// TIA Portal project "FactoryIO_Template_S7-1500_V15_V16" (V16)

(* hardware
DEVICE "S71500/ET200MP-Station_1"  S7-1500 station
   slot 0: "Profilschiene_0"  6ES7 590-1***0-0AA0
   slot 1: "PLC_1"  CPU 1511-1 PN  6ES7 511-1AK00-0AB0  V1.8
   slot 2: "AI 8xU/I/RTD/TC ST_1"  AI 8xU/I/RTD/TC ST  6ES7 531-7KF00-0AB0  V2.0
   slot 3: "AI 8xU/I/RTD/TC ST_2"  AI 8xU/I/RTD/TC ST  6ES7 531-7KF00-0AB0  V2.0
   slot 4: "AI 8xU/I/RTD/TC ST_3"  AI 8xU/I/RTD/TC ST  6ES7 531-7KF00-0AB0  V2.0
   slot 5: "AI 8xU/I/RTD/TC ST_4"  AI 8xU/I/RTD/TC ST  6ES7 531-7KF00-0AB0  V2.0
   slot 6: "DI 16x24VDC BA_1"  DI 16x24VDC BA  6ES7 521-1BH10-0AA0  V1.0
*)

// ===== PLC "PLC_1"  CPU 1511-1 PN =====

VAR_GLOBAL   // PLC tag table "Standard-Variablentabelle"
   "start" AT %E0.0 : Bool;
   "stop" AT %I0.1 : Bool;
   "vsensör" AT %I0.2 : Bool;
   "konveyor1" AT %Q0.0 : Bool;
   "konveyor2" AT %Q0.1 : Bool;
   "itme" AT %Q0.2 : Bool;
   "yr" AT %M0.0 : Bool;
   "itmebant" AT %Q0.3 : Bool;
   "konveyor3" AT %Q0.4 : Bool;
   "itme2" AT %Q0.5 : Bool;
   "itme2bant" AT %Q0.6 : Bool;
   "vsensör2" AT %I0.3 : Bool;
END_VAR

// folder: System blocks/Program resources

DATA_BLOCK "dzr2"   // DB1
{ S7_Optimized_Access := 'TRUE' }
AUTHOR : Simatic
FAMILY : IEC
NAME : IEC_TMR
VERSION : 1.0
// stored: InstanceOfName IEC_TIMER
"IEC_TIMER"
BEGIN
END_DATA_BLOCK

DATA_BLOCK "dzr3"   // DB2
{ S7_Optimized_Access := 'TRUE' }
AUTHOR : Simatic
FAMILY : IEC
NAME : IEC_TMR
VERSION : 1.0
// stored: InstanceOfName IEC_TIMER
"IEC_TIMER"
BEGIN
END_DATA_BLOCK

DATA_BLOCK "dzr1"   // DB3
{ S7_Optimized_Access := 'TRUE' }
AUTHOR : Simatic
FAMILY : IEC
NAME : IEC_TMR
VERSION : 1.0
// stored: InstanceOfName IEC_TIMER
"IEC_TIMER"
BEGIN
END_DATA_BLOCK

// folder: (top level)

FUNCTION "MHJ-PLC-Lab-Function-S71500" : Void   // FC9000, SCL
{ S7_Optimized_Access := 'TRUE' }
VERSION : 0.1
   VAR_TEMP
      Value : Byte;
      ForCounter : Int;
   END_VAR
   VAR CONSTANT
      Value_01_DW : DWord := 16#1223_5486;
      Value_02_DW : DWord := 16#A6C9_D1F5;
   END_VAR
BEGIN

   #Value:=PEEK(area := 16#82,
        dbNumber := 0,
        byteOffset := 511);
   #Value := #Value + 1;

   POKE(area := 16#82,
        dbNumber := 0,
        byteOffset := 511,
        value := #Value);

   POKE(area := 16#82,
        dbNumber := 0,
        byteOffset := 1016,
        value := #Value_01_DW);
   POKE(area := 16#82,
        dbNumber := 0,
        byteOffset := 1020,
        value := #Value_02_DW);

   FOR #ForCounter := 0 TO 63 DO
       #Value:=PEEK(area := 16#1,
            dbNumber := 0,
            byteOffset := #ForCounter);
       POKE(area := 16#81,
            dbNumber := 0,
            byteOffset := #ForCounter,
            value := #Value);
   END_FOR;
   #Value := PEEK(area := 16#1,
                  dbNumber := 0,
                  byteOffset := 512);
   POKE(area := 16#82,
        dbNumber := 0,
        byteOffset := 512,
        value := #Value);
END_FUNCTION

ORGANIZATION_BLOCK "Main"   // OB1, LAD, ProgramCycle
TITLE = "Main Program Sweep (Cycle)"
{ S7_Optimized_Access := 'TRUE' }
VERSION : 0.1
   VAR_INPUT
      Initial_Call : Bool;   // Initial call of this OB
      Remanence : Bool;   // =True, if remanent data are available
   END_VAR
BEGIN

REGION Network 1
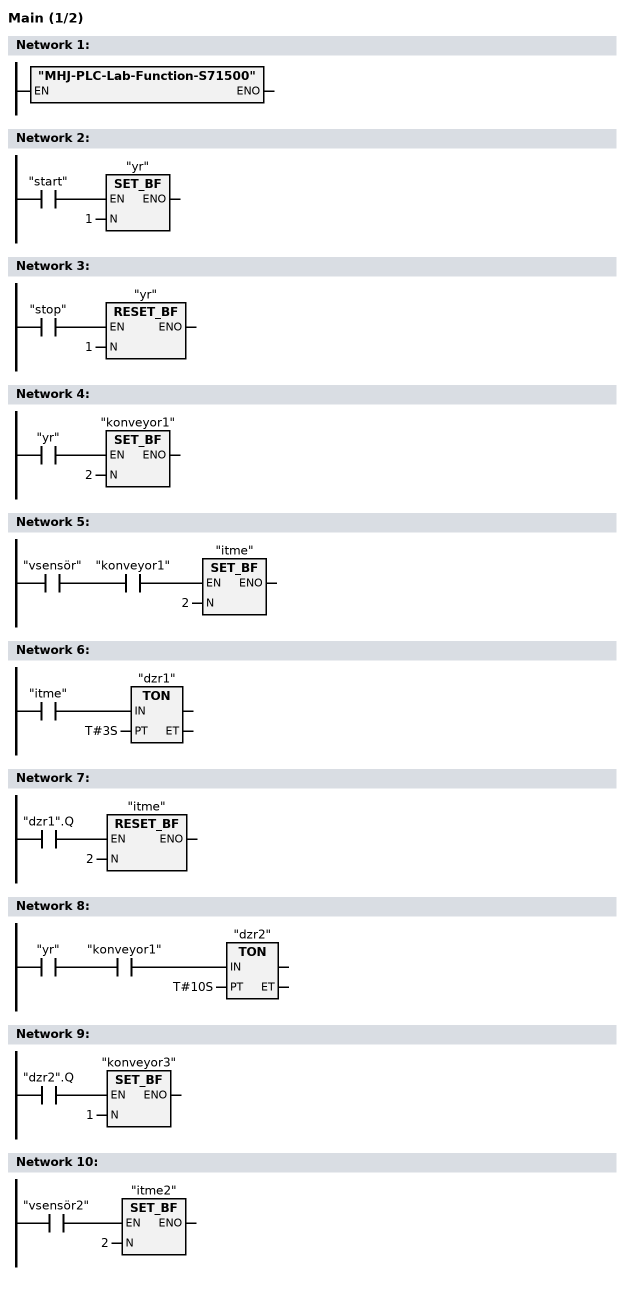
   RUNG wire#powerrail
      "MHJ-PLC-Lab-Function-S71500"()
   END_RUNG
   // the same network as SCL:
   "MHJ-PLC-Lab-Function-S71500"();
END_REGION

REGION Network 2
   // no SCL statement known for SBitfield: written as a call
   IF "start" THEN SET_BF(operand := "yr", n := 1); END_IF;
END_REGION

REGION Network 3
   // no SCL statement known for RBitfield: written as a call
   IF "stop" THEN RESET_BF(operand := "yr", n := 1); END_IF;
END_REGION

REGION Network 4
   // no SCL statement known for SBitfield: written as a call
   IF "yr" THEN SET_BF(operand := "konveyor1", n := 2); END_IF;
END_REGION

REGION Network 5
   // no SCL statement known for SBitfield: written as a call
   IF "vsensör" AND "konveyor1" THEN SET_BF(operand := "itme", n := 2); END_IF;
END_REGION

REGION Network 6
   "dzr1".TON(IN := "itme", PT := T#3S);
END_REGION

REGION Network 7
   // no SCL statement known for RBitfield: written as a call
   IF "dzr1".Q THEN RESET_BF(operand := "itme", n := 2); END_IF;
END_REGION

REGION Network 8
   "dzr2".TON(IN := "yr" AND "konveyor1", PT := T#10S);
END_REGION

REGION Network 9
   // no SCL statement known for SBitfield: written as a call
   IF "dzr2".Q THEN SET_BF(operand := "konveyor3", n := 1); END_IF;
END_REGION

REGION Network 10
   // no SCL statement known for SBitfield: written as a call
   IF "vsensör2" THEN SET_BF(operand := "itme2", n := 2); END_IF;
END_REGION

REGION Network 11
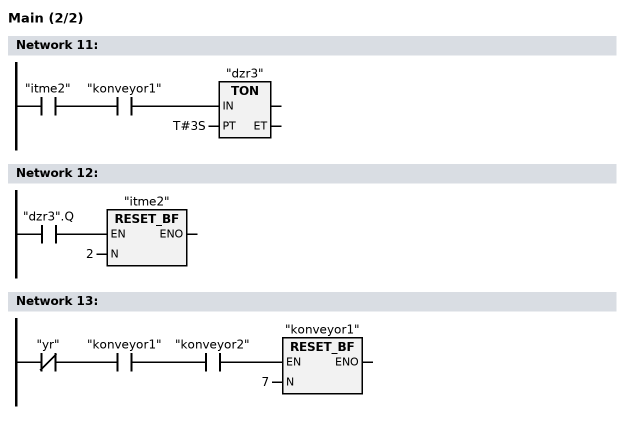
   "dzr3".TON(IN := "itme2" AND "konveyor1", PT := T#3S);
END_REGION

REGION Network 12
   // no SCL statement known for RBitfield: written as a call
   IF "dzr3".Q THEN RESET_BF(operand := "itme2", n := 2); END_IF;
END_REGION

REGION Network 13
   // no SCL statement known for RBitfield: written as a call
   IF NOT "yr" AND "konveyor1" AND "konveyor2" THEN RESET_BF(operand := "konveyor1", n := 7); END_IF;
END_REGION
END_ORGANIZATION_BLOCK